PROGRAM MAIN
VAR

END_VAR

PRG_TerminalMapping.ReadInputs();
PRG_ReadInputs();
PRG_HmiCommands();
PRG_NestSettings();
PRG_HeatStakeProcessSettings();
PRG_StationProcessSettings();
PRG_Main();
PRG_CSV();
PRG_HeatStakeTemperatureSettings();
PRG_Events();
PRG_HmiStatus();
PRG_WriteOutputs();
PRG_TerminalMapping.WriteOutputs();

END_PROGRAM

(* stored: Version 1.1.0.1, ProductVersion 3.1.4026.18
   POU MAIN: Id {58171a7d-5f08-4090-a464-779d1e8200c7}, SpecialFunc None *)
